KUKA KRL program: chk_w7_grp2_opn.src

&ACCESS RVO1
&COMMENT Accelo Traseiro Z2.1_Z2.2
DEF chk_w7_grp2_opn( )

; Check gripper ACCELO TRASEIRO OPEN Z2.1/2
;//---- Start User-------

$TIMER[10] = 0
$TIMER_STOP[10] = FALSE

WAIT FOR (NOT $IN[56] AND NOT $IN[58])
WAIT FOR ($IN[55] AND $IN[57])

$TIMER_STOP[10] = TRUE
$TIMER[10] = 0

;//---- End User---------

END
